TYPE ST_ShopOrderInformation :
STRUCT
	diSo_id                    	: DINT ;
	sSo_number               	: STRING(12) ;
END_STRUCT
END_TYPE

(* stored: Version 1.1.0.1, ProductVersion 3.1.4024.11
   DUT ST_ShopOrderInformation: Id {a1683826-1970-44a6-89b2-d080698769a7} *)
